Fanuc KAREL source: KT00664.KL

PROGRAM KT00664
%NOLOCKGROUP
VAR
  P1: XYZWPR
  P2: XYZWPR
  OUT: INTEGER
BEGIN
  P1.X = 1.0
  P2.Y = 2.0
  P1.X = 1.0
  P2.Y = 2.0
  OUT = + P1
END KT00664
